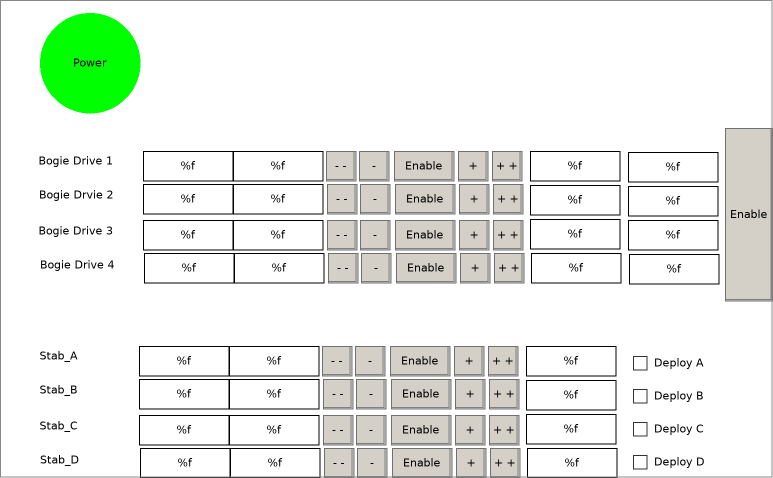
VISUALIZATION Visualization  // 773x478
    Label (25,341 67x30), "Stab_A"
    Rectangle (139,346 90x30), "%f", text variable: GVL.Bogie_Stabiliser_A_Current_Position, colour toggle: GVL.Gripper_In_Position
    Rectangle (229,346 90x30), "%f", text variable: GVL.Bogie_Stabiliser_A_Required_Position
        OnMouseUp: change screen: VisuDialogs.Numpad
    Button (355,346 30x30), "-"
        OnMouseUp: execute { GVL.Bogie_Stabiliser_A_Required_Position := GVL.Bogie_Stabiliser_A_Required_Position - 1; }
    Button (454,346 30x30), "+"
        OnMouseUp: execute { GVL.Bogie_Stabiliser_A_Required_Position := GVL.Bogie_Stabiliser_A_Required_Position + 1; }
    Button (322,346 30x30), "- -"
        OnMouseUp: execute { GVL.Bogie_Stabiliser_A_Required_Position := GVL.Bogie_Stabiliser_A_Required_Position - 10; }
    Button (488,346 30x30), "+ +"
        OnMouseUp: execute { GVL.Bogie_Stabiliser_A_Required_Position := GVL.Bogie_Stabiliser_A_Required_Position + 10; }
    Button (390,346 60x30), "Enable"
        tap GVL.Bogie_Stabiliser_A_Manual_Enable
    Label (25,375 67x30), "Stab_B"
    Rectangle (139,379 90x30), "%f", text variable: GVL.Bogie_Stabiliser_B_Current_Position, colour toggle: GVL.Gripper_In_Position
    Rectangle (229,379 90x30), "%f", text variable: GVL.Bogie_Stabiliser_B_Required_Position
        OnMouseUp: change screen: VisuDialogs.Numpad
    Button (356,379 30x30), "-"
        OnMouseUp: execute { GVL.Bogie_Stabiliser_B_Required_Position := GVL.Bogie_Stabiliser_B_Required_Position - 1; }
    Button (455,379 30x30), "+"
        OnMouseUp: execute { GVL.Bogie_Stabiliser_B_Required_Position := GVL.Bogie_Stabiliser_B_Required_Position + 1; }
    Button (323,379 30x30), "- -"
        OnMouseUp: execute { GVL.Bogie_Stabiliser_B_Required_Position := GVL.Bogie_Stabiliser_B_Required_Position - 10; }
    Button (489,379 30x30), "+ +"
        OnMouseUp: execute { GVL.Bogie_Stabiliser_B_Required_Position := GVL.Bogie_Stabiliser_B_Required_Position + 10; }
    Button (391,379 60x30), "Enable"
        tap GVL.Bogie_Stabiliser_B_Manual_Enable
    Label (25,411 67x30), "Stab_C"
    Rectangle (139,415 90x30), "%f", text variable: GVL.Bogie_Stabiliser_C_Current_Position, colour toggle: GVL.Gripper_In_Position
    Rectangle (229,415 90x30), "%f", text variable: GVL.Bogie_Stabiliser_C_Required_Position
        OnMouseUp: change screen: VisuDialogs.Numpad
    Button (356,415 30x30), "-"
        OnMouseUp: execute { GVL.Bogie_Stabiliser_C_Required_Position := GVL.Bogie_Stabiliser_C_Required_Position - 1; }
    Button (455,415 30x30), "+"
        OnMouseUp: execute { GVL.Bogie_Stabiliser_C_Required_Position := GVL.Bogie_Stabiliser_C_Required_Position + 1; }
    Button (323,415 30x30), "- -"
        OnMouseUp: execute { GVL.Bogie_Stabiliser_C_Required_Position := GVL.Bogie_Stabiliser_C_Required_Position - 10; }
    Button (489,415 30x30), "+ +"
        OnMouseUp: execute { GVL.Bogie_Stabiliser_C_Required_Position := GVL.Bogie_Stabiliser_C_Required_Position + 10; }
    Button (391,415 60x30), "Enable"
        tap GVL.Bogie_Stabiliser_C_Manual_Enable
    Label (26,445 67x30), "Stab_D"
    Rectangle (140,448 90x30), "%f", text variable: GVL.Bogie_Stabiliser_D_Current_Position, colour toggle: GVL.Gripper_In_Position
    Rectangle (230,448 90x30), "%f", text variable: GVL.Bogie_Stabiliser_D_Required_Position
        OnMouseUp: change screen: VisuDialogs.Numpad
    Button (357,448 30x30), "-"
        OnMouseUp: execute { GVL.Bogie_Stabiliser_D_Required_Position := GVL.Bogie_Stabiliser_D_Required_Position - 1; }
    Button (456,448 30x30), "+"
        OnMouseUp: execute { GVL.Bogie_Stabiliser_D_Required_Position := GVL.Bogie_Stabiliser_D_Required_Position + 1; }
    Button (324,448 30x30), "- -"
        OnMouseUp: execute { GVL.Bogie_Stabiliser_D_Required_Position := GVL.Bogie_Stabiliser_D_Required_Position - 10; }
    Button (490,448 30x30), "+ +"
        OnMouseUp: execute { GVL.Bogie_Stabiliser_D_Required_Position := GVL.Bogie_Stabiliser_D_Required_Position + 10; }
    Button (392,448 60x30), "Enable"
        tap GVL.Bogie_Stabiliser_D_Manual_Enable
    Rectangle (526,346 90x30), "%f", text variable: INPUT.Stabilser_A_Torque, colour toggle: GVL.Gripper_In_Position
    Rectangle (526,380 90x30), "%f", text variable: INPUT.Stabilser_B_Torque, colour toggle: GVL.Gripper_In_Position
    Rectangle (526,414 90x30), "%f", text variable: INPUT.Stabilser_C_Torque, colour toggle: GVL.Gripper_In_Position
    Rectangle (527,448 90x30), "%f", text variable: INPUT.Stabilser_D_Torque, colour toggle: GVL.Gripper_In_Position
    Checkbox (631,348 131x30), "Deploy A", variable: GVL.Bogie_Stabiliser_A_Deploy
    Checkbox (631,381 131x30), "Deploy B", variable: GVL.Bogie_Stabiliser_B_Deploy
    Checkbox (631,414 131x30), "Deploy C", variable: GVL.Bogie_Stabiliser_C_Deploy
    Checkbox (631,447 131x30), "Deploy D", variable: GVL.Bogie_Stabiliser_D_Deploy
    Label (29,146 94x30), "Bogie Drive 1"
    Rectangle (143,151 90x30), "%f", text variable: GVL.Bogie_DriveA_Current_Position, colour toggle: GVL.Gripper_In_Position
    Rectangle (233,151 90x30), "%f", text variable: GVL.Bogie_DriveA_Required_Position
        OnMouseUp: change screen: VisuDialogs.Numpad
    Button (359,151 30x30), "-"
        OnMouseUp: execute { GVL.Bogie_DriveA_Required_Position := GVL.Bogie_DriveA_Required_Position - 1; }
    Button (458,151 30x30), "+"
        OnMouseUp: execute { GVL.Bogie_DriveA_Required_Position := GVL.Bogie_DriveA_Required_Position + 1; }
    Button (326,151 30x30), "- -"
        OnMouseUp: execute { GVL.Bogie_DriveA_Required_Position := GVL.Bogie_DriveA_Required_Position - 10; }
    Button (492,151 30x30), "+ +"
        OnMouseUp: execute { GVL.Bogie_DriveA_Required_Position := GVL.Bogie_DriveA_Required_Position + 10; }
    Button (394,151 60x30), "Enable"
        tap GVL.Bogie_DriveA_Manual_Enable
    Label (29,180 95x30), "Bogie Drvie 2"
    Rectangle (143,184 90x30), "%f", text variable: GVL.Bogie_DriveB_Current_Position, colour toggle: GVL.Gripper_In_Position
    Rectangle (233,184 90x30), "%f", text variable: GVL.Bogie_DriveB_Required_Position
        OnMouseUp: change screen: VisuDialogs.Numpad
    Button (360,184 30x30), "-"
        OnMouseUp: execute { GVL.Bogie_DriveB_Required_Position := GVL.Bogie_DriveB_Required_Position - 1; }
    Button (459,184 30x30), "+"
        OnMouseUp: execute { GVL.Bogie_DriveB_Required_Position := GVL.Bogie_DriveB_Required_Position + 1; }
    Button (327,184 30x30), "- -"
        OnMouseUp: execute { GVL.Bogie_DriveB_Required_Position := GVL.Bogie_DriveB_Required_Position - 10; }
    Button (493,184 30x30), "+ +"
        OnMouseUp: execute { GVL.Bogie_DriveB_Required_Position := GVL.Bogie_DriveB_Required_Position + 10; }
    Button (395,184 60x30), "Enable"
        tap GVL.Bogie_DriveB_Manual_Enable p1329445385=TRUE
    Label (29,216 94x30), "Bogie Drive 3"
    Rectangle (143,220 90x30), "%f", text variable: GVL.Bogie_DriveC_Current_Position, colour toggle: GVL.Gripper_In_Position
    Rectangle (233,220 90x30), "%f", text variable: GVL.Bogie_Stabiliser_C_Required_Position
        OnMouseUp: change screen: VisuDialogs.Numpad
    Button (360,220 30x30), "-"
        OnMouseUp: execute { GVL.Bogie_Stabiliser_C_Required_Position := GVL.Bogie_Stabiliser_C_Required_Position - 1; }
    Button (459,220 30x30), "+"
        OnMouseUp: execute { GVL.Bogie_Stabiliser_C_Required_Position := GVL.Bogie_Stabiliser_C_Required_Position + 1; }
    Button (327,220 30x30), "- -"
        OnMouseUp: execute { GVL.Bogie_DriveC_Required_Position := GVL.Bogie_DriveC_Required_Position - 10; }
    Button (493,220 30x30), "+ +"
        OnMouseUp: execute { GVL.Bogie_DriveC_Required_Position := GVL.Bogie_DriveC_Required_Position + 10; }
    Button (395,220 60x30), "Enable"
        tap GVL.Bogie_DriveC_Manual_Enable
    Label (30,250 95x30), "Bogie Drive 4"
    Rectangle (144,253 90x30), "%f", text variable: GVL.Bogie_DriveD_Current_Position, colour toggle: GVL.Gripper_In_Position
    Rectangle (234,253 90x30), "%f", text variable: GVL.Bogie_Stabiliser_D_Required_Position
        OnMouseUp: change screen: VisuDialogs.Numpad
    Button (361,253 30x30), "-"
        OnMouseUp: execute { GVL.Bogie_Stabiliser_D_Required_Position := GVL.Bogie_Stabiliser_D_Required_Position - 1; }
    Button (460,253 30x30), "+"
        OnMouseUp: execute { GVL.Bogie_Stabiliser_D_Required_Position := GVL.Bogie_Stabiliser_D_Required_Position + 1; }
    Button (328,253 30x30), "- -"
        OnMouseUp: execute { GVL.Bogie_DriveD_Required_Position := GVL.Bogie_DriveD_Required_Position - 10; }
    Button (494,253 30x30), "+ +"
        OnMouseUp: execute { GVL.Bogie_Stabiliser_D_Required_Position := GVL.Bogie_Stabiliser_D_Required_Position + 10; }
    Button (396,253 60x30), "Enable"
        tap GVL.Bogie_DriveD_Manual_Enable
    Rectangle (530,151 90x30), "%f", text variable: GVL.Drive_A_Velocity, colour toggle: GVL.Gripper_In_Position
    Rectangle (530,185 90x30), "%f", text variable: GVL.Drive_B_Velocity, colour toggle: GVL.Gripper_In_Position
    Rectangle (530,219 90x30), "%f", text variable: GVL.Drive_C_Velocity, colour toggle: GVL.Gripper_In_Position
    Rectangle (531,253 90x30), "%f", text variable: GVL.Drive_D_Velocity, colour toggle: GVL.Gripper_In_Position
    Button (725,128 48x173), "Enable"
        toggle GVL.DriveAll
    Rectangle (628,152 90x30), "%f", text variable: INPUT.DriveA_Torque, colour toggle: GVL.Gripper_In_Position
    Rectangle (628,186 90x30), "%f", text variable: INPUT.DriveB_Torque, colour toggle: GVL.Gripper_In_Position
    Rectangle (628,220 90x30), "%f", text variable: INPUT.DriveC_Torque, colour toggle: GVL.Gripper_In_Position
    Rectangle (629,254 90x30), "%f", text variable: INPUT.DriveD_Torque, colour toggle: GVL.Gripper_In_Position
    Ellipse (40,13 100x100), "Power", colour toggle: (NOT INPUT.Is_Emergency_Stop_Healthy)
        toggle Input.Is_Emergency_Stop_Healthy
END_VISUALIZATION

(* stored: Version 1.1.0.1, ProductVersion 3.1.4024.4
   Visu Visualization: Id {53bc61be-4496-41fa-87cf-c420270039a6} *)
